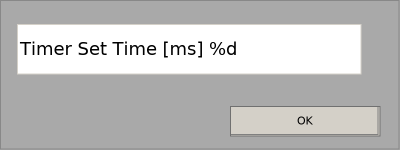
VISUALIZATION DialogTimer_HotWeldValve  // 400x150
    Button (230,106 150x30), "OK"
        OnMouseClick: CloseDialog Dialog=DialogTimer_HotWeldValve, Result=OK, NumpadKeypadSet=True
    Textfield (17,24 344x50), "Timer Set Time [ms] %d", text variable: PersistentStruct.TimeHotWeldPressDown
        OnMouseClick: write the text variable via Edit
END_VISUALIZATION

(* stored: Version 1.1.0.1, ProductVersion 3.1.4024.3
   Visu DialogTimer_HotWeldValve: Id {2c9341d5-6794-445c-a57d-768b3d49264d} *)
